TYPE U_Error_Message :
UNION
END_UNION
END_TYPE

(* stored: Version 1.1.0.1
   DUT U_Error_Message: Id {579d467a-9196-4065-9293-96424004f64e} *)
